(* CODESYS project LibraryRfidReader.library
   Company: Gema
   DefaultNamespace: LibraryRfidReader
   Version: 0.1.1.7
   Placeholder: LibraryRfidReader
   Author: RG
   Description: Functionality of RFID Reader
   Title: RfidReader

Project tree, tasks and I/O mapping:
  libraries: RFID universal data interface TwinCAT, * (Turck); Tc2_Standard, 3.3.3.0 (Beckhoff Automation GmbH); Tc2_System, 3.4.26.0 (Beckhoff Automation GmbH); Tc2_Utilities, 3.3.54.0 (Beckhoff Automation GmbH); Tc3_Module, 3.3.21.0 (Beckhoff Automation GmbH); TcUnit, 1.2.0.0 (www.tcunit.org); TcoCore, 0.11.0.23 (Vortex.Library); TcoData, 0.11.0.23 (Vortex.Library); TcoDrivesBeckhoff, 0.11.0.23 (Vortex.Library); TcoElements, 0.11.0.23 (Vortex.Library); TcoIo, 0.11.0.23 (Vortex.Library); TcoPneumatics, 0.11.0.23 (Vortex.Library)
  DUTs/
  GVLs/
  POUs/
    Context/
      function block MainStation [ST]
      program PRG_TEST [ST]
      function block TcUnitContext [ST]: Main
    Mock/
      function block RfidMockNoRfidInRange [ST]: Execute
      function block RfidMockWorking [ST]: Execute
    Rfid/
      Tasks/
        function block LockTask [ST]: ErrorId, OnAbort, OnDone, OnError, OnStart, Restore, FB_init
        function block ReadDataTask [ST]: Data, ErrorId, OnAbort, OnDone, OnError, OnStart, Restore, FB_init
        function block ReadUidTask [ST]: ErrorId, Uid, OnAbort, OnDone, OnError, OnStart, Restore, FB_init
        function block ResetTask [ST]: ErrorId, OnAbort, OnDone, OnError, OnStart, Restore, FB_init
        function block WriteDataTask [ST]: ErrorId, OnAbort, OnDone, OnError, OnStart, Restore, FB_init
      Wrapper/
        interface IRfidHeadWrapper: Execute
        function block Rfid_FB_Compact_Wrapper [ST]: Execute
      function block RfidHead [ST]: Map, LockMethod, ReadDataMethod, ReadUidMethod, ResetMethod, WriteDataMethod, Data, DataRxLength, Uid, ErrorId, IsError, LockTask, ReadDataTask, ReadUidTask, ResetTask, WriteDataTask, FB_init, Restore, ServiceMode
      data type RfidInOut
    Test/
      function block RfidHead_Test [ST]: ExecuteReadDataNoTagInRange_ExpectErrorWithNoTag, ExecuteReadDataWithOffsetTooHigh_ExpectErrorWithErroId, ExecuteReadDataWithTooLongDataLength_ExpectErrorWithErroId, ExecuteReadDataWrongParameter_ExpectErrorAndStringError, ExecuteReadUidsNoTagInRange_ExpectErrorWithNoTag, Context, EndCycleCount, Environment, Identity, Logger, RealTimeClock, StartCycleCount, ExecuteLock_ExpectStatusDone, ExecuteReadData_ExpectDataAsStringStatusDone, ExecuteReadDataWithOffset_ExpectDataAsString, ExecuteReadUid_ExpectUidAsStringStatusDone, ExecuteReadWriteWithOffset_ExpectStatusDone, ExecuteWriteData_ExpectStatusDone
  Version/
    global variables Global_Version
  VISUs/
*)

// POUs/Rfid/RfidInOut
TYPE
    RfidInOut :
    STRUCT

        myReadData             : ARRAY[0..127] OF BYTE;
        myWriteData            : ARRAY[0..127] OF BYTE;
        xExecute               : BOOL;
        xAbort                 : BOOL;
        udiTimeOut             : UDINT;
        eCommand               : RFID_FB_U.COMMAND;
        udiStartAdress         : UDINT;
        uiDataLenght           : UINT;
        xDone                  : BOOL;
        xBusy                  : BOOL;
        xError                 : BOOL;
        xAborted               : BOOL;
        eErrorID               : RFID_FB_U.ERROR;
        xTP                    : BOOL;
        xRWHeadNotCOnnected    : BOOL;
        uiDataRxLength         : UINT;
        stCompactModeInputMap  : RFID_FB_U.CompactInput_t;
        stCompactModeOutputMap : RFID_FB_U.CompactOutput_t;
    END_STRUCT
END_TYPE

// Version/Global_Version
{attribute 'TcGenerated'}
{attribute 'no-analysis'}
{attribute 'linkalways'}
// This function has been automatically generated from the project information.
VAR_GLOBAL CONSTANT
	{attribute 'const_non_replaced'}
	stLibVersion_RfidReader : ST_LibVersion := (iMajor := 0, iMinor := 1, iBuild := 1, iRevision := 7, nFlags := 0, sVersion := '0.1.1.7');
END_VAR

// POUs/Context/MainStation
FUNCTION_BLOCK MainStation EXTENDS TcoCore.TcoObject
//VAR
//    turckRfidHead : RfidHead(THIS^, T#1MS);
//    sUId          : T_MaxString;
//END_VAR
//VAR
//	    _uid          : BOOL;
//END_VAR

VAR
    rfidHead_Test : RfidHead_Test;

END_VAR

TcUnit.RUN();

END_FUNCTION_BLOCK

// POUs/Rfid/RfidHead
FUNCTION_BLOCK RfidHead EXTENDS TcoCore.TcoComponent
VAR_OUTPUT

END_VAR
VAR
    _itfRfidHeadWrapper : IRfidHeadWrapper;
    _readUidTask        : ReadUidTask(THIS^);
    _readDataTask       : ReadDataTask(THIS^);
    _writeDataTask      : WriteDataTask(THIS^);
    _lockTask           : LockTask(THIS^);
    _resetTask          : ResetTask(THIS^);

    _rfidInOut      : RfidInOut;
    _errorId        : RFID_FB_U.ERROR;
    _uiDataRxLength : UINT;

END_VAR

Map();

_readUidTask(rfidInOut := _rfidInOut, ActionDesc := '<#ReadUid#>');
_readDataTask(rfidInOut := _rfidInOut, ActionDesc := '<#ReadData#>');
_writeDataTask(rfidInOut := _rfidInOut, ActionDesc := '<#WriteData#>');
_lockTask(rfidInOut := _rfidInOut, ActionDesc := '<#WriteData#>');
_resetTask(rfidInOut := _rfidInOut, ActionDesc := '<#ResetTask#>');

METHOD Private Map : BOOL
_itfRfidHeadWrapper.Execute
(
    xExecute              := _rfidInOut.xExecute
    , xAbort              := _rfidInOut.xAbort
    , udiTimeOut          := _rfidInOut.udiTimeOut
    , eCommand            := _rfidInOut.eCommand
    , udiStartAdress      := _rfidInOut.udiStartAdress
    , uiDataLenght        := _rfidInOut.uiDataLenght
    , myWriteData         := _rfidInOut.myWriteData
    , myReadData          => _rfidInOut.myReadData
    , xDone               => _rfidInOut.xDone
    , xBusy               => _rfidInOut.xBusy
    , xError              => _rfidInOut.xError
    , xAborted            => _rfidInOut.xAborted
    , eErrorID            => _rfidInOut.eErrorID
    , xTP                 => _rfidInOut.xTP
    , xRWHeadNotCOnnected => _rfidInOut.xRWHeadNotCOnnected
    , uiDataRxLength      => _rfidInOut.uiDataRxLength
);
END_METHOD

METHOD LockMethod : TcoCore.ITcoTaskStatus
VAR_INPUT
    udiDataLength : UINT; //Length of the Data to read
    StartAdress    : UDINT; // Memory Adress, from which to start
END_VAR
IF (LockTask <> 0) THEN
    _rfidInOut.uiDataLenght   := udiDataLength;
    _rfidInOut.udiStartAdress := StartAdress;
    LockMethod                := LockTask.Invoke();
END_IF
END_METHOD

METHOD ReadDataMethod : TcoCore.ITcoTaskStatus
VAR_INPUT
    udiDataLength : UINT; //Length of the Data to read
    MemoryAddr    : BYTE; // Memory Adress, from which to start
END_VAR
IF (ReadDataTask <> 0) THEN
    _rfidInOut.uiDataLenght   := udiDataLength;
    _rfidInOut.udiStartAdress := MemoryAddr;
    _uiDataRxLength           := _rfidInOut.uiDataRxLength;
    ReadDataMethod            := ReadDataTask.Invoke();
END_IF
END_METHOD

METHOD ReadUidMethod : TcoCore.ITcoTaskStatus
VAR_INPUT
END_VAR
IF (ReadUidTask <> 0) THEN
    ReadUidMethod := ReadUidTask.Invoke();
END_IF
END_METHOD

METHOD ResetMethod : TcoCore.ITcoTaskStatus
IF (ResetTask <> 0) THEN
    ResetMethod := ResetTask.Invoke();
END_IF
END_METHOD

METHOD WriteDataMethod : TcoCore.ITcoTaskStatus
VAR_IN_OUT
    WriteData : ARRAY[*] OF BYTE; //Data to write to Tag
END_VAR
VAR_INPUT
    MemoryAddr : BYTE; // Memory Adress, from which to start
END_VAR
VAR_INST
    _i : DINT;
END_VAR
IF (WriteDataTask <> 0) THEN
    _rfidInOut.uiDataLenght   := SIZEOF(WriteData);
    _rfidInOut.udiStartAdress := MemoryAddr;

    FOR _i := LOWER_BOUND(WriteData, 1) TO UPPER_BOUND(WriteData, 1) DO
        _rfidInOut.myWriteData[_i] := WriteData[_i];
    END_FOR

    _uiDataRxLength := _rfidInOut.uiDataRxLength;
    WriteDataMethod := WriteDataTask.Invoke();
END_IF
END_METHOD

PROPERTY Data : Tc2_System.T_MaxString
GET
Data := _readDataTask.Data;
END_GET
END_PROPERTY

PROPERTY DataRxLength : UINT
GET
DataRxLength := _uiDataRxLength;
END_GET
END_PROPERTY

PROPERTY Uid : Tc2_System.T_MaxString
GET
Uid := _readUidTask.Uid;
END_GET
END_PROPERTY

{attribute 'monitoring' := 'call'}
PROPERTY ErrorId : RFID_FB_U.ERROR
GET
{warning disable C0371}
ErrorId := _readDataTask.ErrorId or _readUidTask.ErrorId or _writeDataTask.ErrorId OR _lockTask.ErrorId;
END_GET
END_PROPERTY

{attribute 'monitoring' := 'call'}
PROPERTY IsError : BOOL
GET
//collected Error from Tasks
IsError := this^.ReadUidTask.Error or this^.ReadDataTask.Error or this^.LockTask.Error or this^.WriteDataTask.Error;
END_GET
END_PROPERTY

PROPERTY LockTask : TcoCore.ITcoTask
GET
LockTask := _lockTask;
END_GET
END_PROPERTY

PROPERTY ReadDataTask : TcoCore.ITcoTask
GET
ReadDataTask := _readDataTask;
END_GET
END_PROPERTY

PROPERTY ReadUidTask : TcoCore.ITcoTask
GET
ReadUidTask := _readUidTask;
END_GET
END_PROPERTY

PROPERTY ResetTask : TcoCore.ITcoTask
GET
ResetTask := _resetTask	;
END_GET
END_PROPERTY

PROPERTY WriteDataTask : TcoCore.ITcoTask
GET
WriteDataTask := _writeDataTask;
END_GET
END_PROPERTY

METHOD FB_init : BOOL
VAR_INPUT
    bInitRetains       : BOOL; // if TRUE, the retain variables are initialized (warm start / cold start)
    bInCopyCode        : BOOL; // if TRUE, the instance afterwards gets moved into the copy code (online change)
    ParentObject       : ITcoObject;
    itfRfidHeadWrapper : IRfidHeadWrapper;
    udiTimeOut         : TIME;
END_VAR
VAR
    _microToMillis : UDINT := 1000;
END_VAR
// This is not clear to me... I from time to time the consumer code does not see 'FB_init' of 'TcoObject', that's why overridden here with super call...
{warning disable C0316}
SUPER^.FB_init(bInitRetains, bInCopyCode, ParentObject);

THIS^._itfRfidHeadWrapper := itfRfidHeadWrapper;

THIS^._rfidInOut.udiTimeOut := TIME_TO_UDINT(udiTimeOut) * _microToMillis;

_readUidTask.FB_init
(
    bInitRetains   := bInitRetains
    , bInCopyCode  := bInCopyCode
    , ParentObject := ParentObject
);
END_METHOD

(*~
    <docu>
        <summary>
            Restore all tasks of this instance into initial state.
        </summary>
    </docu>
~*)
METHOD Restore : ITcoRestorable

IF (ReadUidTask <> 0) THEN
    ReadUidTask.Restore();
END_IF;

IF (ReadDataTask <> 0) THEN
    ReadDataTask.Restore();
END_IF;

IF (WriteDataTask) <> 0 THEN
    WriteDataTask.Restore();
END_IF

IF (LockTask) <> 0 THEN
    LockTask.Restore();
END_IF

IF (ResetTask) <> 0 THEN
    ResetTask.Restore();
END_IF
END_METHOD

METHOD PROTECTED ServiceMode
END_METHOD

END_FUNCTION_BLOCK

// POUs/Rfid/Tasks/ResetTask
FUNCTION_BLOCK ResetTask EXTENDS TcoCore.TcoTask
VAR_IN_OUT
    rfidInOut : RfidInOut;
END_VAR
VAR_INPUT
    ActionDesc : STRING(25);
END_VAR
VAR
    _stringBuilder : TcoCore.StringBuilder;
    _state         : INT;

    _eErrorID   : RFID_FB_U.ERROR;
    _data       : Tc2_System.T_MaxString;
    _noTagFound : BOOL;

    _offSet : UDINT;

    _resetResponseCode : UINT := 16#8000;
END_VAR

IF (THIS^.Execute()) THEN

    CASE _state OF

        10:
            _state := 20;

        20:
            //Command setzen
            rfidInOut.eCommand := RFID_FB_U.COMMAND.RESET;
            _state             := 30;
        30:
            // Start der Operation
            rfidInOut.xExecute := TRUE;

            _state := 40;
        40:
            //            IF rfidInOut.stCompactModeInputMap.eResponseCode = _resetResponseCode THEN
            IF rfidInOut.xDone THEN
                THIS^.DoneWhen(TRUE);
                //                THIS^.Messenger.Info
                //                (
                //                    _stringbuilder.Append('Lock der Daten erfolgreich')
                //                        .Append('Startadresse: ')
                //                        .Append(TO_STRING(rfidinOut.udiStartAdress))
                //                        .Append(' Laenge: ')
                //                        .Append(TO_STRING(rfidInOut.uiDataLenght))
                //                        .ToString()
                //                );

                _state := 0;
            end_IF
    END_CASE
END_IF

{attribute 'monitoring' := 'call'}
PROPERTY ErrorId : RFID_FB_U.ERROR
GET
{warning disable C0371}
ErrorId := _eErrorID;
END_GET
END_PROPERTY

(*~
    <docu>
        <summary>
            Executes when task is aborted.
        </summary>
    </docu>
~*)
METHOD PROTECTED OnAbort
{warning disable C0371}
RfidInOut.eCommand := RFID_FB_U.COMMAND.IDLE;
RfidInOut.xExecute := FALSE;
RfidInOut.xAbort   := FALSE;
END_METHOD

(*~
    <docu>
        <summary>
            Executes when task reaches the ```Done``` state .
        </summary>
    </docu>
~*)
METHOD PROTECTED OnDone
{warning disable C0371}
rfidInOut.xExecute := FALSE;
rfidInOut.eCommand := RFID_FB_U.COMMAND.IDLE;
END_METHOD

(*~
    <docu>
        <summary>
            Executes when task reaches the ```Error``` state.
            <para>
                Do not confuse with <see cref="PlcDocu.TcoCore.TcoTask.WhileError()"/>, that is called cyclically until '''Error''' state is left.
            </para>
        </summary>
    </docu>
~*)
METHOD PROTECTED OnError
{warning disable C0371}
IF _noTagFound THEN
    _eErrorID := RFID_FB_U.ERROR.COMMAND_NO_TAG_FOUND;
    // not implemented by Turck
ELSIF rfidInOut.eErrorID = 16#2901 THEN
    _eErrorID := RFID_FB_U.ERROR.COMMAND_ADDRESS_OUTSIDE_BLOCK_BOUNDARIES;
ELSE
    _eErrorID := rfidInOut.eErrorID;
END_IF

THIS^.Messenger.Build().Append('Rfid Schreib/Lesekopf Fehler : ').Append(to_string(THIS^._eErrorID)).As().AsError();
END_METHOD

(*~
    <docu>
        <summary>
            Executes ones when the task starts (at the moment of transition from the ```Requested``` state into the ```Busy``` state).
        </summary>
    </docu>
~*)
METHOD PROTECTED OnStart
{warning disable C0371}
rfidInOut.eCommand := RFID_FB_U.COMMAND.IDLE;
rfidInOut.xExecute := FALSE;
rfidInOut.xAbort   := FALSE;
_state             := 10;
END_METHOD

(*~
    <docu>
        <summary>
            Restores this instance to the Ready state. Can be called explicitly or from within one of the restore mechanisms.
            <para>
                See also <see cref="PlcDocu.TcoCore.TcoTask.AutoRestorable()"/>
            </para>
        </summary>
    </docu>
~*)
METHOD Restore : ITcoRestorable
{warning disable C0371}
RfidInOut.eCommand := RFID_FB_U.COMMAND.IDLE;
RfidInOut.xExecute := FALSE;
RfidInOut.xAbort   := FALSE;
_noTagFound        := FALSE;
_eErrorID          := RFID_FB_U.ERROR.NO_ERROR;
SUPER^.Restore();
END_METHOD

METHOD PUBLIC FB_init : BOOL
VAR_INPUT
    bInitRetains : BOOL; // if TRUE, the retain variables are initialized (warm start / cold start)
    bInCopyCode  : BOOL; // if TRUE, the instance afterwards gets moved into the copy code (online change)
    ParentObject : ITcoObject;
END_VAR
// This is not clear to me... I from time to time the consumer code does not see 'FB_init' of 'TcoObject', that's why overridden here with super call...
{warning disable C0316}
SUPER^.FB_init(bInitRetains, bInCopyCode, ParentObject);
END_METHOD

END_FUNCTION_BLOCK

// POUs/Rfid/Wrapper/IRfidHeadWrapper
INTERFACE IRfidHeadWrapper

METHOD Execute
VAR_INPUT
    xExecute       : BOOL;
    xAbort         : BOOL;
    udiTimeOut     : UDINT;
    eCommand       : RFID_FB_U.COMMAND;
    udiStartAdress : UDINT;
    uiDataLenght   : UINT;
    myWriteData    : ARRAY[0..127] OF BYTE;
END_VAR
VAR_OUTPUT
    myReadData          : ARRAY[0..127] OF BYTE;
    xDone               : BOOL;
    xBusy               : BOOL;
    xError              : BOOL;
    xAborted            : BOOL;
    eErrorID            : RFID_FB_U.ERROR;
    xTP                 : BOOL;
    xRWHeadNotCOnnected : BOOL;
    uiDataRxLength      : UINT;
END_VAR
END_METHOD

END_INTERFACE

// POUs/Rfid/Tasks/ReadUidTask
FUNCTION_BLOCK ReadUidTask EXTENDS TcoCore.TcoTask
VAR_IN_OUT
    rfidInOut : RfidInOut;
END_VAR
VAR_INPUT
    ActionDesc : STRING(25);
END_VAR

VAR
    _stringBuilder : TcoCore.StringBuilder;
    _state         : INT;
    _coding        : ARRAY[0..7] OF BYTE;
    _index         : INT;
    _hex           : Tc2_System.T_MaxString := '16# ';
    _uidDataLength : UINT                   := 8;

    _eErrorID   : RFID_FB_U.ERROR;
    _noTagFound : BOOL;
    _uid        : Tc2_System.T_MaxString;
END_VAR

IF (THIS^.Execute()) THEN
    THIS^.ThrowWhen(rfidInOut.xError);

    CASE _state OF

        10:
            // Tag vorhanden
            IF NOT rfidInOut.xTP THEN
                THIS^.Messenger.Error
                (
                    _stringBuilder.Append(ActionDesc)
                        .Append('Tag nicht vorhanden bei Leseversuch')
                        .ToString()
                );

                _noTagFound := TRUE;
                ThrowWhen(TRUE);
            ELSE
                _state := 20;
            END_IF
        20:
            //Command setzen
            rfidInOut.eCommand     := command.INVENTORY;
            rfidInOut.uiDataLenght := _uidDataLength;
            _state                 := 30;
        30:
            // Start der Operation
            rfidInOut.xExecute := TRUE;
            _uid               := '';

            _state := 40;
        40:
            // Warte auf Ende Operation
            rfidInOut.myReadData[_index] :=
                (THIS^.rfidInOut.myReadData[_index]);

            IF rfidInOut.xError THEN
                _uid := '--Error--';
            ELSIF rfidInOut.xDone THEN
                FOR _index := 0 TO UINT_TO_INT(rfidInOut.uiDataLenght - 1) DO

                    _uid := Concat
                    (
                        _uid
                        , BYTE_TO_HEXSTR(in := rfidInOut.myReadData[_index], iPrecision := 2, bLoCase := FALSE)
                    );
                END_FOR

                THIS^.DoneWhen(rfidInOut.xDone);
                THIS^.Messenger.Info('Lesen UID erfolgreich');
                _state := 0;
            END_IF
    END_CASE
END_IF

{attribute 'monitoring' := 'call'}
PROPERTY ErrorId : RFID_FB_U.ERROR
GET
{warning disable C0371}
ErrorId := _eErrorID;
END_GET
END_PROPERTY

PROPERTY Uid : Tc2_System.T_MaxString
GET
Uid := _uId;
END_GET
END_PROPERTY

(*~
    <docu>
        <summary>
            Executes when task is aborted.
        </summary>
    </docu>
~*)
METHOD PROTECTED OnAbort
{warning disable C0371}
RfidInOut.eCommand := RFID_FB_U.COMMAND.IDLE;
RfidInOut.xExecute := FALSE;
RfidInOut.xAbort   := FALSE;
END_METHOD

(*~
    <docu>
        <summary>
            Executes when task reaches the ```Done``` state .
        </summary>
    </docu>
~*)
METHOD PROTECTED OnDone
{warning disable C0371}
rfidInOut.xExecute := FALSE;
rfidInOut.eCommand := RFID_FB_U.COMMAND.IDLE;
END_METHOD

(*~
    <docu>
        <summary>
            Executes when task reaches the ```Error``` state.
            <para>
                Do not confuse with <see cref="PlcDocu.TcoCore.TcoTask.WhileError()"/>, that is called cyclically until '''Error''' state is left.
            </para>
        </summary>
    </docu>
~*)
METHOD PROTECTED OnError
{warning disable C0371}

IF _noTagFound THEN
    _eErrorID := RFID_FB_U.ERROR.COMMAND_NO_TAG_FOUND;
ELSE
    _eErrorID := rfidInOut.eErrorID;
END_IF

THIS^.Messenger.Build().Append('Rfid Schreib/Lesekopf Fehler : ').Append(to_string(THIS^._eErrorID)).As().AsError();
END_METHOD

(*~
    <docu>
        <summary>
            Executes ones when the task starts (at the moment of transition from the ```Requested``` state into the ```Busy``` state).
        </summary>
    </docu>
~*)
METHOD PROTECTED OnStart
{warning disable C0371}
rfidInOut.eCommand := RFID_FB_U.COMMAND.IDLE;
rfidInOut.xExecute := FALSE;
rfidInOut.xAbort   := FALSE;
_state             := 10;
END_METHOD

(*~
    <docu>
        <summary>
            Restores this instance to the Ready state. Can be called explicitly or from within one of the restore mechanisms.
            <para>
                See also <see cref="PlcDocu.TcoCore.TcoTask.AutoRestorable()"/>
            </para>
        </summary>
    </docu>
~*)
METHOD Restore : ITcoRestorable
{warning disable C0371}
RfidInOut.eCommand := RFID_FB_U.COMMAND.IDLE;
RfidInOut.xExecute := FALSE;
RfidInOut.xAbort   := FALSE;
_eErrorID          := RFID_FB_U.ERROR.NO_ERROR;
SUPER^.Restore();
END_METHOD

METHOD PUBLIC FB_init : BOOL
VAR_INPUT
    bInitRetains : BOOL; // if TRUE, the retain variables are initialized (warm start / cold start)
    bInCopyCode  : BOOL; // if TRUE, the instance afterwards gets moved into the copy code (online change)
    ParentObject : ITcoObject;
END_VAR
// This is not clear to me... I from time to time the consumer code does not see 'FB_init' of 'TcoObject', that's why overridden here with super call...
{warning disable C0316}
SUPER^.FB_init(bInitRetains, bInCopyCode, ParentObject);
END_METHOD

END_FUNCTION_BLOCK

// POUs/Rfid/Tasks/ReadDataTask
FUNCTION_BLOCK ReadDataTask EXTENDS TcoCore.TcoTask
VAR_IN_OUT
    rfidInOut : RfidInOut;
END_VAR
VAR_INPUT
    ActionDesc : STRING(25);
END_VAR
VAR
    _stringBuilder : TcoCore.StringBuilder;
    _state         : INT;
    _coding        : ARRAY[0..3] OF BYTE;
    _index         : INT;
    _hex           : Tc2_System.T_MaxString := '16#';

    _eErrorID   : RFID_FB_U.ERROR;
    _data       : Tc2_System.T_MaxString;
    _noTagFound : BOOL;
END_VAR

IF (THIS^.Execute()) THEN
    THIS^.ThrowWhen(rfidInOut.xError);

    CASE _state OF

        10:
            // Tag vorhanden
            IF NOT rfidInOut.xTP THEN
                THIS^.Messenger.Error
                (
                    _stringBuilder.Append(ActionDesc)
                        .Append('Tag nicht vorhanden bei Leseversuch')
                        .ToString()
                );

                _noTagFound := true;
                ThrowWhen(TRUE);
            ELSE
                _state := 20;
            END_IF
        20:
            //Command setzen
            rfidInOut.eCommand := RFID_FB_U.COMMAND.READ;
            _state             := 30;
        30:
            // Start der Operation
            rfidInOut.xExecute := TRUE;
            _data              := '';

            _state := 40;
        40:
            // Warte auf Ende Operation
            IF rfidInOut.xError THEN
                 _data              := '--Error--';
            ELSIF rfidInOut.xDone THEN
                FOR _index := 0 TO UINT_TO_INT(rfidInOut.uiDataLenght - 1) DO
                    rfidInOut.myReadData[_index] :=
                        (THIS^.rfidInOut.myReadData[_index]);

                    _data := Concat
                    (
                        _data
                        , Concat
                        (
                            ' '
                            , BYTE_TO_HEXSTR(in := rfidInOut.myReadData[_index], iPrecision := 2, bLoCase := FALSE)
                        )
                    );
                END_FOR

                _data := Concat(_hex, _data);

                THIS^.DoneWhen(rfidInOut.xDone);
                THIS^.Messenger.Info('Lesen der Daten erfolgreich');
                _state := 0;
            END_IF
    END_CASE
END_IF

PROPERTY Data : Tc2_System.T_MaxString
GET
Data := _data;
END_GET
END_PROPERTY

{attribute 'monitoring' := 'call'}
PROPERTY ErrorId : RFID_FB_U.ERROR
GET
{warning disable C0371}
ErrorId := _eErrorID;
END_GET
END_PROPERTY

(*~
    <docu>
        <summary>
            Executes when task is aborted.
        </summary>
    </docu>
~*)
METHOD PROTECTED OnAbort
{warning disable C0371}
RfidInOut.eCommand := RFID_FB_U.COMMAND.IDLE;
RfidInOut.xExecute := FALSE;
RfidInOut.xAbort   := FALSE;
END_METHOD

(*~
    <docu>
        <summary>
            Executes when task reaches the ```Done``` state .
        </summary>
    </docu>
~*)
METHOD PROTECTED OnDone
{warning disable C0371}
rfidInOut.xExecute := FALSE;
rfidInOut.eCommand := RFID_FB_U.COMMAND.IDLE;
END_METHOD

(*~
    <docu>
        <summary>
            Executes when task reaches the ```Error``` state.
            <para>
                Do not confuse with <see cref="PlcDocu.TcoCore.TcoTask.WhileError()"/>, that is called cyclically until '''Error''' state is left.
            </para>
        </summary>
    </docu>
~*)
METHOD PROTECTED OnError
{warning disable C0371}
IF _noTagFound THEN
    _eErrorID := RFID_FB_U.ERROR.COMMAND_NO_TAG_FOUND;
ELSE
    _eErrorID := rfidInOut.eErrorID;
END_IF

THIS^.Messenger.Build().Append('Rfid Schreib/Lesekopf Fehler : ').Append(to_string(THIS^._eErrorID)).As().AsError();
END_METHOD

(*~
    <docu>
        <summary>
            Executes ones when the task starts (at the moment of transition from the ```Requested``` state into the ```Busy``` state).
        </summary>
    </docu>
~*)
METHOD PROTECTED OnStart
{warning disable C0371}
rfidInOut.eCommand := RFID_FB_U.COMMAND.IDLE;
rfidInOut.xExecute := FALSE;
rfidInOut.xAbort   := FALSE;
_state             := 10;
END_METHOD

(*~
    <docu>
        <summary>
            Restores this instance to the Ready state. Can be called explicitly or from within one of the restore mechanisms.
            <para>
                See also <see cref="PlcDocu.TcoCore.TcoTask.AutoRestorable()"/>
            </para>
        </summary>
    </docu>
~*)
METHOD Restore : ITcoRestorable
{warning disable C0371}
RfidInOut.eCommand := RFID_FB_U.COMMAND.IDLE;
RfidInOut.xExecute := FALSE;
RfidInOut.xAbort   := FALSE;
_noTagFound        := FALSE;
_eErrorID          := RFID_FB_U.ERROR.NO_ERROR;
SUPER^.Restore();
END_METHOD

METHOD PUBLIC FB_init : BOOL
VAR_INPUT
    bInitRetains : BOOL; // if TRUE, the retain variables are initialized (warm start / cold start)
    bInCopyCode  : BOOL; // if TRUE, the instance afterwards gets moved into the copy code (online change)
    ParentObject : ITcoObject;
END_VAR
// This is not clear to me... I from time to time the consumer code does not see 'FB_init' of 'TcoObject', that's why overridden here with super call...
{warning disable C0316}
SUPER^.FB_init(bInitRetains, bInCopyCode, ParentObject);
END_METHOD

END_FUNCTION_BLOCK

// POUs/Rfid/Tasks/WriteDataTask
FUNCTION_BLOCK WriteDataTask EXTENDS TcoCore.TcoTask
VAR_IN_OUT
    rfidInOut : RfidInOut;
END_VAR
VAR_INPUT
    ActionDesc : STRING(25);
END_VAR
VAR
    _stringBuilder : TcoCore.StringBuilder;
    _state         : INT;

    _eErrorID   : RFID_FB_U.ERROR;
    _data       : Tc2_System.T_MaxString;
    _noTagFound : BOOL;

    _offSet : UDINT;
END_VAR

IF (THIS^.Execute()) THEN
    THIS^.ThrowWhen(rfidInOut.xError);

    CASE _state OF

        10:
            // Tag vorhanden
            IF NOT rfidInOut.xTP THEN
                THIS^.Messenger.Error
                (
                    _stringBuilder.Append(ActionDesc)
                        .Append('Tag nicht vorhanden bei Schreibversuch')
                        .ToString()
                );

                _noTagFound := true;
                ThrowWhen(TRUE);
            ELSE
                _state := 20;
            END_IF
        20:
            //Command setzen
            _offSet            := rfidInOut.udiStartAdress;
            rfidInOut.eCommand := RFID_FB_U.COMMAND.WRITE;
            _state             := 30;
        30:
            // Start der Operation
            rfidInOut.xExecute := TRUE;
            _data              := '';

            _state := 40;
        40:
            // Warte auf Ende Operation
            IF rfidInOut.xError THEN
                ;
            ELSIF rfidInOut.xDone THEN

                THIS^.DoneWhen(rfidInOut.xDone);
                THIS^.Messenger.Info('Schreiben der Daten erfolgreich');
                _state := 0;
            END_IF
    END_CASE
END_IF

{attribute 'monitoring' := 'call'}
PROPERTY ErrorId : RFID_FB_U.ERROR
GET
{warning disable C0371}
ErrorId := _eErrorID;
END_GET
END_PROPERTY

(*~
    <docu>
        <summary>
            Executes when task is aborted.
        </summary>
    </docu>
~*)
METHOD PROTECTED OnAbort
{warning disable C0371}
RfidInOut.eCommand := RFID_FB_U.COMMAND.IDLE;
RfidInOut.xExecute := FALSE;
RfidInOut.xAbort   := FALSE;
END_METHOD

(*~
    <docu>
        <summary>
            Executes when task reaches the ```Done``` state .
        </summary>
    </docu>
~*)
METHOD PROTECTED OnDone
{warning disable C0371}
rfidInOut.xExecute := FALSE;
rfidInOut.eCommand := RFID_FB_U.COMMAND.IDLE;
END_METHOD

(*~
    <docu>
        <summary>
            Executes when task reaches the ```Error``` state.
            <para>
                Do not confuse with <see cref="PlcDocu.TcoCore.TcoTask.WhileError()"/>, that is called cyclically until '''Error''' state is left.
            </para>
        </summary>
    </docu>
~*)
METHOD PROTECTED OnError
{warning disable C0371}
IF _noTagFound THEN
    _eErrorID := RFID_FB_U.ERROR.COMMAND_NO_TAG_FOUND;
ELSE
    _eErrorID := rfidInOut.eErrorID;
END_IF

THIS^.Messenger.Build().Append('Rfid Schreib/Lesekopf Fehler : ').Append(to_string(THIS^._eErrorID)).As().AsError();
END_METHOD

(*~
    <docu>
        <summary>
            Executes ones when the task starts (at the moment of transition from the ```Requested``` state into the ```Busy``` state).
        </summary>
    </docu>
~*)
METHOD PROTECTED OnStart
{warning disable C0371}
rfidInOut.eCommand := RFID_FB_U.COMMAND.IDLE;
rfidInOut.xExecute := FALSE;
rfidInOut.xAbort   := FALSE;
_state             := 10;
END_METHOD

(*~
    <docu>
        <summary>
            Restores this instance to the Ready state. Can be called explicitly or from within one of the restore mechanisms.
            <para>
                See also <see cref="PlcDocu.TcoCore.TcoTask.AutoRestorable()"/>
            </para>
        </summary>
    </docu>
~*)
METHOD Restore : ITcoRestorable
{warning disable C0371}
RfidInOut.eCommand := RFID_FB_U.COMMAND.IDLE;
RfidInOut.xExecute := FALSE;
RfidInOut.xAbort   := FALSE;
_noTagFound        := FALSE;
_eErrorID          := RFID_FB_U.ERROR.NO_ERROR;
SUPER^.Restore();
END_METHOD

METHOD PUBLIC FB_init : BOOL
VAR_INPUT
    bInitRetains : BOOL; // if TRUE, the retain variables are initialized (warm start / cold start)
    bInCopyCode  : BOOL; // if TRUE, the instance afterwards gets moved into the copy code (online change)
    ParentObject : ITcoObject;
END_VAR
// This is not clear to me... I from time to time the consumer code does not see 'FB_init' of 'TcoObject', that's why overridden here with super call...
{warning disable C0316}
SUPER^.FB_init(bInitRetains, bInCopyCode, ParentObject);
END_METHOD

END_FUNCTION_BLOCK

// POUs/Rfid/Tasks/LockTask
FUNCTION_BLOCK LockTask EXTENDS TcoCore.TcoTask
VAR_IN_OUT
    rfidInOut : RfidInOut;
END_VAR
VAR_INPUT
    ActionDesc : STRING(25);
END_VAR
VAR
    _stringBuilder : TcoCore.StringBuilder;
    _state         : INT;

    _eErrorID   : RFID_FB_U.ERROR;
    _data       : Tc2_System.T_MaxString;
    _noTagFound : BOOL;

    _offSet : UDINT;
END_VAR

IF (THIS^.Execute()) THEN
    THIS^.ThrowWhen(rfidInOut.xError);

    CASE _state OF

        10:
            // Tag vorhanden
            IF NOT rfidInOut.xTP THEN
                THIS^.Messenger.Error
                (
                    _stringBuilder.Append(ActionDesc)
                        .Append('Tag nicht vorhanden bei Schreibversuch')
                        .ToString()
                );

                _noTagFound := true;
                ThrowWhen(TRUE);
            ELSE
                _state := 20;
            END_IF
        20:
            //Command setzen
            rfidInOut.eCommand := RFID_FB_U.COMMAND.SET_PERMA_LOCK;
            ADSLOGSTR
            (
                msgCtrlMask := ADSLOG_MSGTYPE_ERROR
                , msgFmtStr := 'Startadresse bei CMD: %s'
                , strArg    := TO_STRING(rfidInOut.udiStartAdress)
            );

            _state := 30;
        30:
            // Start der Operation
            rfidInOut.xExecute := TRUE;

            _state := 40;
        40:
            // Warte auf Ende Operation
            IF rfidInOut.xError THEN
                ;
            ELSIF rfidInOut.xDone THEN

                THIS^.DoneWhen(rfidInOut.xDone);
                //                THIS^.Messenger.Info
                //                (
                //                    _stringbuilder.Append('Lock der Daten erfolgreich')
                //                        .Append('Startadresse: ')
                //                        .Append(TO_STRING(rfidinOut.udiStartAdress))
                //                        .Append(' Laenge: ')
                //                        .Append(TO_STRING(rfidInOut.uiDataLenght))
                //                        .ToString()
                //                );
                ADSLOGSTR
                (
                    msgCtrlMask := ADSLOG_MSGTYPE_ERROR
                    , msgFmtStr := 'Startadresse nach Done: %s'
                    , strArg    := TO_STRING(rfidInOut.udiStartAdress)
                );

                _state := 0;
            END_IF
    END_CASE
END_IF

{attribute 'monitoring' := 'call'}
PROPERTY ErrorId : RFID_FB_U.ERROR
GET
{warning disable C0371}
ErrorId := _eErrorID;
END_GET
END_PROPERTY

(*~
    <docu>
        <summary>
            Executes when task is aborted.
        </summary>
    </docu>
~*)
METHOD PROTECTED OnAbort
{warning disable C0371}
RfidInOut.eCommand := RFID_FB_U.COMMAND.IDLE;
RfidInOut.xExecute := FALSE;
RfidInOut.xAbort   := FALSE;
END_METHOD

(*~
    <docu>
        <summary>
            Executes when task reaches the ```Done``` state .
        </summary>
    </docu>
~*)
METHOD PROTECTED OnDone
{warning disable C0371}
rfidInOut.xExecute := FALSE;
rfidInOut.eCommand := RFID_FB_U.COMMAND.IDLE;
END_METHOD

(*~
    <docu>
        <summary>
            Executes when task reaches the ```Error``` state.
            <para>
                Do not confuse with <see cref="PlcDocu.TcoCore.TcoTask.WhileError()"/>, that is called cyclically until '''Error''' state is left.
            </para>
        </summary>
    </docu>
~*)
METHOD PROTECTED OnError
{warning disable C0371}
IF _noTagFound THEN
    _eErrorID := RFID_FB_U.ERROR.COMMAND_NO_TAG_FOUND;
    // not implemented by Turck
ELSIF rfidInOut.eErrorID = 16#2901 THEN
    _eErrorID := RFID_FB_U.ERROR.COMMAND_ADDRESS_OUTSIDE_BLOCK_BOUNDARIES;
ELSE
    _eErrorID := rfidInOut.eErrorID;
END_IF

THIS^.Messenger.Build().Append('Rfid Schreib/Lesekopf Fehler : ').Append(to_string(THIS^._eErrorID)).As().AsError();
END_METHOD

(*~
    <docu>
        <summary>
            Executes ones when the task starts (at the moment of transition from the ```Requested``` state into the ```Busy``` state).
        </summary>
    </docu>
~*)
METHOD PROTECTED OnStart
{warning disable C0371}
rfidInOut.eCommand := RFID_FB_U.COMMAND.IDLE;
rfidInOut.xExecute := FALSE;
rfidInOut.xAbort   := FALSE;
_state             := 10;
END_METHOD

(*~
    <docu>
        <summary>
            Restores this instance to the Ready state. Can be called explicitly or from within one of the restore mechanisms.
            <para>
                See also <see cref="PlcDocu.TcoCore.TcoTask.AutoRestorable()"/>
            </para>
        </summary>
    </docu>
~*)
METHOD Restore : ITcoRestorable
{warning disable C0371}
RfidInOut.eCommand := RFID_FB_U.COMMAND.IDLE;
RfidInOut.xExecute := FALSE;
RfidInOut.xAbort   := FALSE;
_noTagFound        := FALSE;
_eErrorID          := RFID_FB_U.ERROR.NO_ERROR;
SUPER^.Restore();
END_METHOD

METHOD PUBLIC FB_init : BOOL
VAR_INPUT
    bInitRetains : BOOL; // if TRUE, the retain variables are initialized (warm start / cold start)
    bInCopyCode  : BOOL; // if TRUE, the instance afterwards gets moved into the copy code (online change)
    ParentObject : ITcoObject;
END_VAR
// This is not clear to me... I from time to time the consumer code does not see 'FB_init' of 'TcoObject', that's why overridden here with super call...
{warning disable C0316}
SUPER^.FB_init(bInitRetains, bInCopyCode, ParentObject);
END_METHOD

END_FUNCTION_BLOCK

// POUs/Test/RfidHead_Test
FUNCTION_BLOCK RfidHead_Test EXTENDS TcUnit.FB_TestSuite IMPLEMENTS TcoCore.ITcoContext
VAR
    //Context for TcOpen
    _nfContext : TcoCore.TcoContextNfCompatibility;
END_VAR
VAR
    _wrapper_RfidMockNoRfidInRange : RfidMockNoRfidInRange;

    sut_readDataNoTag                  : RfidHead(THIS^, _wrapper_RfidMockNoRfidInRange, T#10MS);
    sut_readUidNoTag                   : RfidHead(THIS^, _wrapper_RfidMockNoRfidInRange, T#10MS);
    _wrapper_readUid                   : RfidMockWorking;
    sut_readUidSuccess                 : RfidHead(THIS^, _wrapper_readUid, T#10MS);
    _wrapper_readData                  : RfidMockWorking;
    sut_readDataSuccess                : RfidHead(THIS^, _wrapper_readData, T#10MS);
    _wrapper_RfidMockTooLong           : RfidMockWorking;
    sut_readDataTooLongString          : RfidHead(THIS^, _wrapper_RfidMockTooLong, T#10MS);
    _wrapper_writeData                 : RfidMockWorking;
    sut_writeDataSuccess               : RfidHead(THIS^, _wrapper_writeData, T#10MS);
    _wrapper_readDataWithOffset        : RfidMockWorking;
    sut_readDataWithOffset             : RfidHead(THIS^, _wrapper_readDataWithOffset, T#10MS);
    _wrapper_writeDataWithOffset       : RfidMockWorking;
    sut_writeDataWithOffsetSuccess     : RfidHead(THIS^, _wrapper_writeDataWithOffset, T#10MS);
    _wrapper_readDataWithOffsetTooLong : RfidMockWorking;
    sut_readDataWithOffsetTooLong      : RfidHead(THIS^, _wrapper_readDataWithOffsetTooLong, T#10MS);
    _wrapper_lock                      : RfidMockWorking;
    sut_lockSuccess                    : RfidHead(THIS^, _wrapper_lock, T#10MS);
    _wrapper_RfidMockCreateError           : RfidMockWorking;
    sut_readDataCreateEmptyString         : RfidHead(THIS^, _wrapper_RfidMockCreateError, T#10MS);


END_VAR

_nfContext.VolatileOpen(); //Required for TCopen
//==============================================

//
ExecuteReadDataWithTooLongDataLength_ExpectErrorWithErroId();
ExecuteReadDataWithOffsetTooHigh_ExpectErrorWithErroId();
//
ExecuteReadUidsNoTagInRange_ExpectErrorWithNoTag();
ExecuteReadDataNoTagInRange_ExpectErrorWithNoTag();

//
ExecuteReadUid_ExpectUidAsStringStatusDone();
ExecuteReadData_ExpectDataAsStringStatusDone();
ExecuteReadDataWithOffset_ExpectDataAsString();

//
ExecuteWriteData_ExpectStatusDone();
ExecuteReadDataWrongParameter_ExpectErrorAndStringError();
// Lock testen,
// Locken, muss Status done, Schreiben mit Error
ExecuteLock_ExpectStatusDone();
//==============================================
_nfContext.VolatileClose();

METHOD PRIVATE ExecuteReadDataNoTagInRange_ExpectErrorWithNoTag
VAR_INST
    _udiDataLength : uINT := 3;
    _result        : BOOL;
    _firstRun      : BOOL := TRUE;

    _expectedErrorId : RFID_FB_U.ERROR;
    _errorId         : RFID_FB_U.ERROR;

END_VAR
TcUnit.TEST('ExecuteReadDataNoTagInRange_ExpectErrorWithNoTag');

//Assert Initial State
_result := FALSE;

IF _firstRun THEN
    _firstRun := FALSE;
    THIS^.
        AssertEquals_BOOL
    (
        _result
        , sut_readDataNoTag.ReadDataMethod(_udiDataLength, 0).Error
        , 'No Error should be Start Parameter'
    );
END_IF

//Arrange
sut_readDataNoTag();

//Act, Use ReadDataMethod()
sut_readDataNoTag.ReadDataMethod(_udiDataLength, 0);

IF sut_readDataNoTag.isError THEN
    //Assert
    _result := TRUE;

    AssertEquals_BOOL
    (
        _result
        , sut_readDataNoTag.ReadDataMethod(_udiDataLength, 0).Error
        , 'Method did not throw Error'
    );

    AssertEquals_BOOL
    (
        _result
        , sut_readDataNoTag.ReadDataTask.Error
        , 'Task did not throw Error'
    );

    _errorId         := sut_readDataNoTag.ErrorId;
    _expectedErrorId := RFID_FB_U.ERROR.COMMAND_NO_TAG_FOUND;
    AssertEquals(Expected := _expectedErrorId, Actual := _errorId, Message := 'ErrorId must match (No Tag Found)!');

    //Act, Restore(), Error shall disappear
    sut_readDataNoTag.Restore();
    _result := FALSE;

    AssertEquals_BOOL
    (
        _result
        , sut_readDataNoTag.ReadDataTask.Error
        , 'Reset did not Work, Still Status Error'
    );

    _errorId         := sut_readDataNoTag.ErrorId;
    _expectedErrorId := RFID_FB_U.ERROR.NO_ERROR;

    AssertEquals_BOOL
    (
        _result
        , sut_readDataNoTag.ReadDataTask.Error
        , 'Reset did not Work, ErrorID ahs to be No_Error'
    );

    TcUnit.TEST_FINISHED();
END_IF
END_METHOD

METHOD PRIVATE ExecuteReadDataWithOffsetTooHigh_ExpectErrorWithErroId
VAR_INST
    _udiDataLength : UINT := 4;
    _offSet        : BYTE := 120;
    _result        : BOOL;
    _firstRun      : BOOL := TRUE;

    _expectedErrorId : RFID_FB_U.ERROR;
    _errorId         : RFID_FB_U.ERROR;

END_VAR
TcUnit.TEST('ExecuteReadDataWithOffsetTooHigh_ExpectErrorWithErroId');
//28 blocks, 4 bytes each, => 112 bytes max user Memory!

//Arrange
sut_readDataWithOffsetTooLong();

//Act, Use ReadDataMethod()
sut_readDataWithOffsetTooLong.ReadDataMethod(udiDataLength := _udiDataLength, MemoryAddr := _offSet);

IF sut_readDataWithOffsetTooLong.ReadDataTask.Error
       OR sut_readUidNoTag.ReadDataTask.Done THEN

    //Assert

    _expectedErrorId := ERROR.COMMAND_ADDRESS_OUTSIDE_TAG_SPECS;
    _errorId         := sut_readDataWithOffsetTooLong.ErrorId;
    AssertEquals(Expected := _expectedErrorId, Actual := _errorId, Message := 'ErrorId must match!');

    _result := TRUE;
    AssertEquals_BOOL
    (
        _result
        , sut_readDataWithOffsetTooLong.ReadDataMethod(_udiDataLength, 0).Error
        , 'Method must throw Error'
    );

    AssertEquals_BOOL
    (
        _result
        , sut_readDataWithOffsetTooLong.ReadDataTask.Error
        , 'Task did not throw Error'
    );

    AssertEquals_BOOL
    (
        _result
        , sut_readDataWithOffsetTooLong.isError
        , 'FB must throw Error'
    );

    //Act, Restore(), Error shall disappear
    sut_readDataWithOffsetTooLong.Restore();
    // more Cycles needed
    sut_readDataWithOffsetTooLong();
    sut_readDataWithOffsetTooLong();
    sut_readDataWithOffsetTooLong();

    _result := FALSE;

    AssertEquals_BOOL
    (
        _result
        , sut_readDataWithOffsetTooLong.IsError
        , 'Reset did not Work, Still Status Error'
    );

    _errorId         := sut_readDataWithOffsetTooLong.ErrorId;
    _expectedErrorId := RFID_FB_U.ERROR.NO_ERROR;
    AssertEquals(Expected := _expectedErrorId, Actual := _errorId, Message := 'ErrorId must match (No Error)!');

    TcUnit.TEST_FINISHED();
END_IF
END_METHOD

METHOD PRIVATE ExecuteReadDataWithTooLongDataLength_ExpectErrorWithErroId
VAR_INST
    _udiDataLength : uINT := 113;
    _result        : BOOL;
    _firstRun      : BOOL := TRUE;

    _expectedErrorId : RFID_FB_U.ERROR;
    _errorId         : RFID_FB_U.ERROR;

END_VAR
TcUnit.TEST('ExecuteReadDataWithTooLongDataLength_ExpectErrorWithErroId');
//28 blocks, 4 bytes each, => 112 bytes max user Memory!

//Arrange
sut_readDataTooLongString();

//Act, Use ReadDataMethod()
sut_readDataTooLongString.ReadDataMethod(udiDataLength := _udiDataLength, MemoryAddr := 0);

IF sut_readDataTooLongString.ReadDataTask.Error
       OR sut_readUidNoTag.ReadDataTask.Done THEN

    //Assert

    _expectedErrorId := ERROR.COMMAND_LENGTH_OUTSIDE_TAG_SPECS;
    _errorId         := sut_readDataTooLongString.ErrorId;
    AssertEquals(Expected := _expectedErrorId, Actual := _errorId, Message := 'ErrorId must match!');

    _result := TRUE;
    AssertEquals_BOOL
    (
        _result
        , sut_readDataTooLongString.ReadDataMethod(_udiDataLength, 0).Error
        , 'Method must throw Error'
    );

    AssertEquals_BOOL
    (
        _result
        , sut_readDataTooLongString.ReadDataTask.Error
        , 'Task did not throw Error'
    );

    AssertEquals_BOOL
    (
        _result
        , sut_readDataTooLongString.isError
        , 'FB must throw Error'
    );

    //Act, Restore(), Error shall disappear
    sut_readDataTooLongString.Restore();
    // more Cycles needed
    sut_readDataTooLongString();
    sut_readDataTooLongString();
    sut_readDataTooLongString();

    _result := FALSE;

    AssertEquals_BOOL
    (
        _result
        , sut_readDataTooLongString.IsError
        , 'Reset did not Work, Still Status Error'
    );

    _errorId         := sut_readDataTooLongString.ErrorId;
    _expectedErrorId := RFID_FB_U.ERROR.NO_ERROR;
    AssertEquals(Expected := _expectedErrorId, Actual := _errorId, Message := 'ErrorId must match (No Error)!');

    TcUnit.TEST_FINISHED();
END_IF
END_METHOD

METHOD ExecuteReadDataWrongParameter_ExpectErrorAndStringError
VAR_INST
    _udiDataLength : UINT := 4;
    _offSet        : BYTE := 120;
    _result        : BOOL;
    _resultString  : STRING := '--Error--';
    _firstRun      : BOOL := TRUE;

    _expectedErrorId : RFID_FB_U.ERROR;
    _errorId         : RFID_FB_U.ERROR;

END_VAR
TcUnit.TEST('ExecuteReadDataWrongParameter_ExpectErrorAndStringError');

sut_readDataCreateEmptyString();

//Act, Use ReadDataMethod()
sut_readDataCreateEmptyString.ReadDataMethod(udiDataLength := _udiDataLength, MemoryAddr := _offSet);

IF sut_readDataCreateEmptyString.ReadDataTask.Error THEN
    //Assert

    _result := TRUE;
    AssertEquals_BOOL
    (
        _result
        , sut_readDataCreateEmptyString.ReadDataMethod(_udiDataLength, 0).Error
        , 'Method must throw Error'
    );

    AssertEquals_STRING
    (
        Expected  := _resultString
        , actual  := sut_readDataCreateEmptyString.Data
        , Message := 'Data String muss --Error-- sein '
    );

    TcUnit.TEST_FINISHED();
END_IF
END_METHOD

METHOD PRIVATE ExecuteReadUidsNoTagInRange_ExpectErrorWithNoTag
VAR_INST
    _udiDataLength : INT := 10;
    _result        : BOOL;
    _firstRun      : BOOL := TRUE;

    _errorId         : RFID_FB_U.ERROR;
    _expectedErrorId : RFID_FB_U.ERROR;

END_VAR
TcUnit.TEST('ExecuteReadUidMethodNoTagInRange_ExpectErrorWithTimeOut');

//Assert Initial State
_result := FALSE;

IF _firstRun THEN
    _firstRun := FALSE;
    THIS^.
        AssertEquals_BOOL
    (
        _result
        , sut_readUidNoTag.ReadUidMethod().Error
        , 'No Error should be Start Parameter'
    );
END_IF

//Arrange
sut_readUidNoTag();

//Act, Use ReadUidMethod()
IF sut_readUidNoTag.ReadUidMethod().Error
       OR sut_readUidNoTag.ReadUidMethod().Done THEN
    //Assert
    _result := TRUE;

    AssertEquals_BOOL
    (
        _result
        , sut_readUidNoTag.ReadUidMethod().Error
        , 'Method did not throw Error'
    );

    AssertEquals_BOOL
    (
        _result
        , sut_readUidNoTag.ReadUidTask.Error
        , 'Task did not throw Error'
    );

    _errorId         := sut_readUidNoTag.ErrorId;
    _expectedErrorId := RFID_FB_U.ERROR.COMMAND_NO_TAG_FOUND;
    AssertEquals(Expected := _expectedErrorId, Actual := _errorId, Message := 'ErrorId must match (No Tag Found)!');

    //Act, Restore(), Error shall disappear
    sut_readUidNoTag.Restore();
    _result := FALSE;

    AssertEquals_BOOL
    (
        _result
        , sut_readUidNoTag.ReadUidTask.Error
        , 'Reset did not Work, Still Status Error'
    );

    TcUnit.TEST_FINISHED();
END_IF
END_METHOD

PROPERTY Context : TcoCore.ITcoContext
GET
Context := This^._nfContext;
END_GET
END_PROPERTY

PROPERTY EndCycleCount : ULINT
GET
EndCycleCount := THIS^._nfContext._endCycleCount;
END_GET
END_PROPERTY

PROPERTY Environment : TcoCore.ITcoContextEnvironment
GET
Environment := THIS^._nfContext._settings;
END_GET
END_PROPERTY

PROPERTY Identity : ULINT
GET
Identity := THIS^._nfContext._Identity;
END_GET
END_PROPERTY

PROPERTY Logger : TcoCore.ITcoLogger
GET
Logger := THIS^._nfContext._logger;
END_GET
END_PROPERTY

PROPERTY RealTimeClock : TcoCore.ITcoRtc
GET
RealTimeClock := THIS^._nfContext._rtc;
END_GET
END_PROPERTY

PROPERTY StartCycleCount : ULINT
GET
StartCycleCount := THIS^._nfContext._startCycleCount;
END_GET
END_PROPERTY

METHOD PRIVATE ExecuteLock_ExpectStatusDone
VAR_INST
    _udiDataLength : UINT := 4;
    _offSet        : BYTE := 1;
    _result        : BOOL;

    _first : BOOL := TRUE;
END_VAR
TcUnit.TEST('ExecuteLock_ExpectStatusDone');
//Arrange
sut_lockSuccess();

//Act
sut_lockSuccess.LockMethod(udiDataLength := _udiDataLength, StartAdress := _offSet);

_result := TRUE;

//Needs two Cycles to get from Status Requested to Buisy (TcOpen Framework)
sut_lockSuccess();

IF _first THEN
    AssertEquals_BOOL
    (
        Expected  := _result
        , Actual  := sut_lockSuccess.LockTask.Busy
        , Message := 'Status Busy muss true sein'
    );

    _first := FALSE;
END_IF

IF sut_lockSuccess.LockTask.Done THEN

    _result := FALSE;
    AssertEquals_BOOL
    (
        Expected  := _result
        , Actual  := sut_lockSuccess.LockTask.Busy
        , Message := 'Status Busy muss false sein'
    );

    _result := TRUE;
    AssertEquals_BOOL
    (
        Expected  := _result
        , Actual  := sut_lockSuccess.LockMethod(udiDataLength := _udiDataLength, StartAdress := _offSet).Done
        , Message := 'Status Done muss true sein'
    );

    TcUnit.TEST_FINISHED();
END_IF
END_METHOD

METHOD PRIVATE ExecuteReadData_ExpectDataAsStringStatusDone
VAR_INST
    _data          : T_MaxString;
    _expectedData  : T_MaxString := '16# 05 06 07 08';
    _result        : BOOL;
    _udiDataLength : uINT := 4;
END_VAR
//{warning disable C0371}
TcUnit.TEST('ExecuteReadData_ExpectDataAsStringStatusDone');
//Arrange
sut_readDataSuccess();

//Act

sut_readDataSuccess.ReadDataMethod(_udiDataLength, 0);
//Assert

IF sut_readDataSuccess.ReadDataTask.Done THEN
    _data := sut_readDataSuccess.Data;

    AssertEquals_STRING(Expected := _expectedData, Actual := _data, Message := 'Daten passt nicht');

    //Busy off
    _result := FALSE;
    AssertEquals_BOOL
    (
        Expected  := _result
        , Actual  := sut_readDataSuccess.ReadDataTask.Busy
        , Message := 'Status Busy muss false sein'
    );

    //Status Done mus True sein
    _result := true;
    AssertEquals_BOOL
    (
        Expected  := _result
        , Actual  := sut_readDataSuccess.ReadDataMethod(_udiDataLength, 0).Done
        , Message := 'Status Done muss true sein'
    );

    //Status Done false again
    sut_readDataSuccess.Restore();
    _result := FALSE;
    AssertEquals_BOOL
    (
        Expected  := _result
        , Actual  := sut_readDataSuccess.ReadDataMethod(_udiDataLength, 0).Done
        , Message := 'Status Done muss false sein nach Reset'
    );

    TcUnit.TEST_FINISHED();
END_IF
END_METHOD

METHOD PRIVATE ExecuteReadDataWithOffset_ExpectDataAsString
VAR_INST
    _data          : T_MaxString;
    _expectedData  : T_MaxString := '16# 06 07 08 09'; // Ohne '16# 05 06 07 08' => mit 16# 06 07 08 00
    _result        : BOOL;
    _udiDataLength : uINT  := 4;
    _offSet        : BYTE := 1;
END_VAR
//{warning disable C0371}
TcUnit.TEST('ExecuteReadDataWithOffset_ExpectDataAsString');
//Arrange
sut_readDataWithOffset();

//Act

sut_readDataWithOffset.ReadDataMethod(_udiDataLength, _offSet);
//Assert

IF sut_readDataWithOffset.ReadDataTask.Done THEN
    _data := sut_readDataWithOffset.Data;

    AssertEquals_STRING(Expected := _expectedData, Actual := _data, Message := 'Daten passt nicht');

    //Busy off
    _result := FALSE;
    AssertEquals_BOOL
    (
        Expected  := _result
        , Actual  := sut_readDataWithOffset.ReadDataTask.Busy
        , Message := 'Status Busy muss false sein'
    );

    //Status Done mus True sein
    _result := true;
    AssertEquals_BOOL
    (
        Expected  := _result
        , Actual  := sut_readDataWithOffset.ReadDataMethod(_udiDataLength, _offSet).Done
        , Message := 'Status Done muss true sein'
    );

    //Status Done false again
    sut_readDataWithOffset.Restore();
    _result := FALSE;
    AssertEquals_BOOL
    (
        Expected  := _result
        , Actual  := sut_readDataWithOffset.ReadDataTask.Done
        , Message := 'Status Done muss false sein nach Reset'
    );

    TcUnit.TEST_FINISHED();
END_IF
END_METHOD

METHOD PRIVATE ExecuteReadUid_ExpectUidAsStringStatusDone
VAR_INST
    _uId         : T_MaxString;
    _expectedUid : T_MaxString := 'E0040150ACF4F3AD';
    _result      : BOOL;
END_VAR
TcUnit.TEST('ExecuteReadUid_ExpectUidAsStringStatusDone');
//Arrange
sut_readUidSuccess();

//Act

sut_readUidSuccess.ReadUidMethod();
//Assert

IF sut_readUidSuccess.ReadUidTask.Done THEN
    _uId := sut_readUidSuccess.Uid;

    AssertEquals_STRING(Expected := _expectedUid, Actual := _uId, Message := 'UID passt nicht');

    //Busy off
    _result := FALSE;
    AssertEquals_BOOL
    (
        Expected  := _result
        , Actual  := sut_readUidSuccess.ReadUidMethod().Busy
        , Message := 'Status Busy muss false sein'
    );

    //Status Done mus True sein
    _result := true;
    AssertEquals_BOOL
    (
        Expected  := _result
        , Actual  := sut_readUidSuccess.ReadUidMethod().Done
        , Message := 'Status Done muss true sein'
    );

    //Status Done false again
    sut_readUidSuccess.Restore();
    _result := FALSE;
    AssertEquals_BOOL
    (
        Expected  := _result
        , Actual  := sut_readUidSuccess.ReadUidMethod().Done
        , Message := 'Status Done muss false sein nach Reset'
    );

    TcUnit.TEST_FINISHED();
END_IF
END_METHOD

METHOD PRIVATE ExecuteReadWriteWithOffset_ExpectStatusDone
VAR_INST
    _data          : T_MaxString;
    _expectedData  : T_MaxString := '16# 06 07 08 00'; // Ohne '16# 05 06 07 08' => mit 16# 06 07 08 00
    _result        : BOOL;
    _udiDataLength : uINT  := 4;
    _offSet        : BYTE := 1;
END_VAR
//{warning disable C0371}
TcUnit.TEST('ExecuteReadWriteWithOffset_ExpectStatusDone');
//Arrange
sut_writeDataWithOffsetSuccess();

//Act

sut_writeDataWithOffsetSuccess.ReadDataMethod(_udiDataLength, _offSet);
//Assert

IF sut_writeDataWithOffsetSuccess.ReadDataTask.Done THEN
    _data := sut_writeDataWithOffsetSuccess.Data;

    AssertEquals_STRING(Expected := _expectedData, Actual := _data, Message := 'Daten passt nicht');

    //Busy off
    _result := FALSE;
    AssertEquals_BOOL
    (
        Expected  := _result
        , Actual  := sut_writeDataWithOffsetSuccess.ReadDataTask.Busy
        , Message := 'Status Busy muss false sein'
    );

    //Status Done mus True sein
    _result := true;
    AssertEquals_BOOL
    (
        Expected  := _result
        , Actual  := sut_writeDataWithOffsetSuccess.ReadDataMethod(_udiDataLength, _offSet).Done
        , Message := 'Status Done muss true sein'
    );

    //Status Done false again
    sut_writeDataWithOffsetSuccess.Restore();
    _result := FALSE;
    AssertEquals_BOOL
    (
        Expected  := _result
        , Actual  := sut_writeDataWithOffsetSuccess.ReadDataTask.Done
        , Message := 'Status Done muss false sein nach Reset'
    );

    TcUnit.TEST_FINISHED();
END_IF
END_METHOD

METHOD PRIVATE ExecuteWriteData_ExpectStatusDone
VAR_INST
    _testArray : ARRAY[0..4] OF BYTE;

    _result : BOOL;

    _first  : BOOL := TRUE;
    _offSet : BYTE := 1;
END_VAR
TcUnit.TEST('ExecuteWriteData_ExpectStatusDone');
//Arrange
sut_writeDataSuccess();

//Act
sut_writeDataSuccess.WriteDataMethod(WriteData := _testArray, MemoryAddr := 0);

_result := TRUE;

//Needs two Cycles to get from Status Requested to Buisy (TcOpen Framework)
sut_writeDataSuccess();

IF _first THEN
    AssertEquals_BOOL
    (
        Expected  := _result
        , Actual  := sut_writeDataSuccess.WriteDataTask.Busy
        , Message := 'Status Busy muss true sein'
    );

    _first := FALSE;
END_IF

IF sut_writeDataSuccess.WriteDataTask.Done THEN

    _result := FALSE;
    AssertEquals_BOOL
    (
        Expected  := _result
        , Actual  := sut_writeDataSuccess.WriteDataTask.Busy
        , Message := 'Status Busy muss false sein'
    );

    _result := TRUE;
    AssertEquals_BOOL
    (
        Expected  := _result
        , Actual  := sut_writeDataSuccess.WriteDataMethod(WriteData := _testArray, MemoryAddr := 0).Done
        , Message := 'Status Done muss true sein'
    );

    TcUnit.TEST_FINISHED();
END_IF
END_METHOD

END_FUNCTION_BLOCK

// POUs/Mock/RfidMockNoRfidInRange
FUNCTION_BLOCK RfidMockNoRfidInRange IMPLEMENTS IRfidHeadWrapper
VAR
    _timeOut        : Tc2_Standard.TON;
    _executionTimer : Tc2_Standard.TON;

    _udintToMillis : UDINT := 1000;
    _busy          : BOOL;

END_VAR

METHOD Execute
VAR_INPUT
    xExecute               : BOOL;
    xAbort                 : BOOL;
    udiTimeOut             : UDINT;
    eCommand               : RFID_FB_U.COMMAND;
    udiStartAdress         : UDINT;
    uiDataLenght           : UINT;
    myWriteData            : ARRAY[0..127] OF BYTE;
END_VAR
VAR_OUTPUT
    myReadData            : ARRAY[0..127] OF BYTE;
    xDone                 : BOOL;
    xBusy                 : BOOL;
    xError                : BOOL;
    xAborted              : BOOL;
    eErrorID              : RFID_FB_U.ERROR;
    xTP                   : BOOL;
    xRWHeadNotCOnnected   : BOOL;
    uiDataRxLength        : UINT;
END_VAR
IF xExecute THEN
    _busy := TRUE;
END_IF

//28 blocks, 4 bytes each, => 112 bytes max user Memory!
uiDataRxLength := uiDataLenght;
xBusy          := _busy;

_timeOut(in := _busy, PT := UDINT_TO_TIME(udiTimeOut) / _udintToMillis);

xTP := FALSE;

IF _timeOut.Q THEN
    xBusy    := FALSE;
    xError   := TRUE;
    eErrorId := RFID_FB_U.ERROR.TIME_OUT;
END_IF
END_METHOD

END_FUNCTION_BLOCK

// POUs/Mock/RfidMockWorking
FUNCTION_BLOCK RfidMockWorking IMPLEMENTS IRfidHeadWrapper
VAR
    _timeOut        : Tc2_Standard.TON;
    _executionTimer : Tc2_Standard.TON := (PT := _executionTime);
    _executionTime  : TIME             := t#5ms;

    _udIntToMillis : UDINT := 1000;

    _resultUid : ARRAY[0..7] OF BYTE :=
    [
        16#E0
        , 16#04
        , 16#01
        , 16#50
        , 16#AC
        , 16#F4
        , 16#F3
        , 16#AD
    ];

    _states :
        (Idle
        , Busy
        , ElectedMethod
        , ReadUid
        , ReadData
        , WriteData
        , Error
        , Restore);
    _index : INT;

    _rfidInOut : RfidInOut;
END_VAR

{warning disable C0371}
//28 blocks, 4 bytes each, => 112 bytes max user Memory!

CASE _states OF
    Idle:
        _rfidInOut.xbusy := _rfidInOut.xExecute;
        _rfidInOut.xTP   := TRUE;

        IF _rfidInOut.xbusy THEN
            _states := Busy;
        END_IF

    Busy:

        _rfidInOut.uiDataRxLength := _rfidInOut.uiDataLenght;
        _timeOut(in := _rfidInOut.xbusy, PT := UDINT_TO_TIME(_rfidInOut.udiTimeOut) / _udintToMillis);
        _executionTimer(in := _rfidInOut.xBusy);

        IF _timeOut.Q THEN
            _states             := Error;
            _rfidInOut.eErrorID := RFID_FB_U.ERROR.TIME_OUT;
            RETURN;

        ELSIF _executionTimer.Q THEN
            _states := ElectedMethod;
        END_IF

    ElectedMethod:
        IF _rfidInOut.uiDataLenght > 112 THEN
            _states             := Error;
            _rfidInOut.eErrorID := RFID_FB_U.ERROR.COMMAND_LENGTH_OUTSIDE_TAG_SPECS;
            RETURN;
        ELSIF _rfidInOut.udiStartAdress > 112 THEN
            _states             := Error;
            _rfidInOut.eErrorID := RFID_FB_U.ERROR.COMMAND_ADDRESS_OUTSIDE_TAG_SPECS;
            RETURN;
        END_IF

        IF _rfidInOut.eCommand = RFID_FB_U.COMMAND.INVENTORY THEN
            FOR _index := 0 TO 7 DO
                _rfidInOut.myReadData[_index] := _resultUid[_index];
            END_FOR

            _rfidInOut.xbusy := FALSE;
            _rfidInOut.xDone := TRUE;
        ELSIF _rfidInOut.eCommand = RFID_FB_U.COMMAND.READ THEN

            FOR _index := 0 TO UINT_TO_INT(_rfidInOut.uiDataLenght) - 1 DO
                _rfidInOut.myReadData[_index] := 16#05 + INT_TO_BYTE(_index + UDINT_TO_INT(_rfidInOut.udiStartAdress));
            END_FOR

            _rfidInOut.xbusy := FALSE;
            _rfidInOut.xDone := TRUE; //

        ELSIF _rfidInOut.eCommand = RFID_FB_U.COMMAND.WRITE THEN
            _rfidInOut.xbusy := FALSE;
            _rfidInOut.xDone := TRUE;

        ELSIF _rfidInOut.eCommand = RFID_FB_U.COMMAND.SET_PERMA_LOCK THEN
            _rfidInOut.xbusy := FALSE;
            _rfidInOut.xDone := TRUE;
        END_IF

    Error:
        _executionTimer(in := FALSE);
        _timeOut(in := FALSE);
        _rfidInOut.xbusy  := FALSE;
        _rfidInOut.xError := TRUE;

        IF NOT _rfidInOut.xExecute THEN
            _States := Restore;
        END_IF
    Restore:
        _rfidInOut.xDone    := FALSE;
        _rfidInOut.xError   := FALSE;
        _rfidInOut.eErrorID := RFID_FB_U.ERROR.NO_ERROR;
        _States             := Idle;
END_CASE

METHOD Execute
VAR_INPUT
    xExecute               : BOOL;
    xAbort                 : BOOL;
    udiTimeOut             : UDINT := 10000;
    eCommand               : RFID_FB_U.COMMAND;
    udiStartAdress         : UDINT;
    uiDataLenght           : UINT;
    myWriteData            : ARRAY[0..127] OF BYTE;
END_VAR
VAR_OUTPUT
    myReadData            : ARRAY[0..127] OF BYTE;
    xDone                 : BOOL;
    xBusy                 : BOOL;
    xError                : BOOL;
    xAborted              : BOOL;
    eErrorID              : RFID_FB_U.ERROR;
    xTP                   : BOOL;
    xRWHeadNotCOnnected   : BOOL;
    uiDataRxLength        : UINT;
END_VAR
VAR_INST
    _busy : BOOL;
END_VAR
THIS^();

_rfidInOut.xExecute       := xExecute;
_rfidInOut.xAbort         := xAbort;
_rfidInOut.udiTimeOut     := udiTimeOut;
_rfidInOut.eCommand       := eCommand;
_rfidInOut.udiStartAdress := udiStartAdress;
_rfidInOut.uiDataLenght   := uiDataLenght;
_rfidInOut.myWriteData    := myWriteData;

myReadData          := _rfidInOut.myReadData;
xDone               := _rfidInOut.xDone;
xBusy               := _rfidInOut.xBusy;
xError              := _rfidInOut.xError;
xAborted            := _rfidInOut.xAborted;
eErrorID            := _rfidInOut.eErrorID;
xTP                 := _rfidInOut.xTP;
xRWHeadNotCOnnected := _rfidInOut.xRWHeadNotCOnnected;
uiDataRxLength      := _rfidInOut.uiDataRxLength;
END_METHOD

END_FUNCTION_BLOCK

// POUs/Context/PRG_TEST
PROGRAM PRG_TEST
VAR
    _testSuite : TcUnitContext;
END_VAR

_testSuite.Run();
_testSuite.RtcSynchronize(true, '', 60);

END_PROGRAM

// POUs/Context/TcUnitContext
FUNCTION_BLOCK TcUnitContext EXTENDS TcoCore.TcoContext
VAR
    _mainStation : MainStation(THIS^);

    {attribute addProperty Name "Versionsnummer Plc"}
    _sVersion : STRING(23);
    //~
    _stProgramVersion : ST_LibVersion;
    //~

END_VAR

(*~
    <docu>
        <summary>
            Main method of the TcoContext. This is the entry point of any control logic that belongs to this context.
            The call of this method is ensured by calling the <c>InstanceName.Run()</c> method, and it must not be called explicitly.
            This method is abstract, and it must be overridden in derived block.
        </summary>
    </docu>
~*)
METHOD PROTECTED Main

_mainStation();
END_METHOD

END_FUNCTION_BLOCK

// POUs/Rfid/Wrapper/Rfid_FB_Compact_Wrapper
FUNCTION_BLOCK Rfid_FB_Compact_Wrapper IMPLEMENTS IRfidHeadWrapper
VAR
    //Instantiate the function block
    turckRfid : RFID_FB_U.FB_Compact;

    // Create mapping to the I/O data of the corresponding channel
    stCompactModeInputMap  AT %I* : RFID_FB_U.CompactInput_t;
    stCompactModeOutputMap AT %Q* : RFID_FB_U.CompactOutput_t;
    // The Rx & Tx data mapping shown below is for example purposes only.
    // The actual array size can be 8,16,32,64 or 128 depending on slot configuration of the TBEC-LL-4RFID-8DXP box in the IO tree
    abyRxDataMapCompactMode AT %I* : ARRAY[0..127] OF BYTE;
    abyTxDataMapCompactMode AT %Q* : ARRAY[0..127] OF BYTE;
END_VAR

METHOD Execute
VAR_INPUT
    xExecute               : BOOL;
    xAbort                 : BOOL;
    udiTimeOut             : UDINT;
    eCommand               : RFID_FB_U.COMMAND;
    udiStartAdress         : UDINT;
    uiDataLenght           : UINT;
    myWriteData            : ARRAY[0..127] OF BYTE;
END_VAR
VAR_OUTPUT
    myReadData            : ARRAY[0..127] OF BYTE;
    xDone                 : BOOL;
    xBusy                 : BOOL;
    xError                : BOOL;
    xAborted              : BOOL;
    eErrorID              : RFID_FB_U.ERROR;
    xTP                   : BOOL;
    xRWHeadNotCOnnected   : BOOL;
    uiDataRxLength        : UINT;
END_VAR
turckRfid
(
    xExecute              := xExecute
    , xAbort              := xAbort
    , udiTimeOut          := udiTimeOut
    , xDone               => xDone
    , xBusy               => xBusy
    , xError              => xError
    , xAborted            => xAborted
    , eCommand            := eCommand
    , rStatusMapping      := stCompactModeInputMap
    , rControlMapping     := stCompactModeOutputMap
    , udiStartAddress     := udiStartAdress
    , uiDataLength        := uiDataLenght
    , eErrorID            => eErrorID
    , xTP                 => xTP
    , xRWHeadNotConnected => xRWHeadNotCOnnected
    , uiDataRxLength      => uiDataRxLength
    , pReadDataMapping    := abyRxDataMapCompactMode
    , pWriteDataMapping   := abyTxDataMapCompactMode
    , pDataTx             := myWriteData
    , pDataRx             := myReadData
);
END_METHOD

END_FUNCTION_BLOCK
